GLOBALCONSTANTS AID_CO (* Container object attribute ids *)
  (* Standard: 61499-1; Description: Copyright (c) 2023 HR Agrartechnik GmbH This program and the accompanying materials are made available under the terms of the Eclipse Public License 2.0 which is available at https://www.eclipse.org/legal/epl-2.0/ SPDX-License-Identifier: EPL-2.0 *)
  (* Version 1.0, 2026-06-20, Franz Höpfinger, HR Agrartechnik GmbH *)
  PACKAGE isobus::UT::Q::const::AID;
  VAR_GLOBAL CONSTANT
    WIDTH : USINT := USINT#1; (* 1: AID_CO_WIDTH - Maximum width of the container's area in pixels. Objects or portions outside *)
    HEIGHT : USINT := USINT#2; (* 2: AID_CO_HEIGHT - Maximum height of the container's area in pixels. Objects or portions outside *)
    HIDDEN : USINT := USINT#3; (* 3: AID_CO_HIDDEN - 0 = FALSE, 1 = TRUE. Indicates whether or not this container and its child *)
  END_VAR
END_GLOBALCONSTANTS
